{attribute 'call_after_init'}
FUNCTION_BLOCK FB_AmphosShutterEnable_Test EXTENDS FB_TestSuite
VAR_INPUT
END_VAR
VAR_OUTPUT
END_VAR
VAR
END_VAR

LocksWithHardwareFailure();
LocksWithLOCOLeak();
LocksWithLOTAOLeak();
LocksWithLUTLeak();
LocksWithAmphosOnAndTemperatureEvent01();
LocksWithAmphosOnAndTemperatureEvent02();
LocksWithAmphosOnAndTemperatureEvent03();
LocksWithAmphosOnAndTemperatureEvent04();
LocksWithTempMonError01();
LocksWithTempMonError02();
LocksWithTempMonError03();
LocksWithTempMonError04();
LocksWithTempMonError05();
LocksWithTempMonError06();
LocksWithTempMonError07();
LocksWithTempMonError08();
LocksWithOpcpaCriticalError();
LocksWithDumpChillerError();
LocksWithMRCError02();
LocksWithMRCError03();
EnablesWithAmphosOffAndTemperatureEvent01();
EnablesWithAmphosOffAndTemperatureEvent02();
EnablesWithAmphosOffAndTemperatureEvent03();
EnablesWithAmphosOffAndTemperatureEvent04();
EnablesWithTemperatureEventOverride01();
EnablesWithTemperatureEventOverride02();
EnablesWithTemperatureEventOverride03();
EnablesWithTemperatureEventOverride04();
EnablesWithOpcpaMinorError();
EnablesWhenNoError();

METHOD EnablesWhenNoError
VAR
	stErrors : st_ErrorStates;
	stOpcpaSetpoints : ST_LaserSetpoints := F_LaserSetpoints();
	bResult : BOOL;
END_VAR
TEST('EnablesWhenNoError');

bResult := F_AmphosShutterEnable(
	bAmphosOn := TRUE, 
	fOpcpaVoltage := stOpcpaSetpoints.nMinNominalVoltage, 
	bLoopTempOverride01 := FALSE,
	bLoopTempOverride02 := FALSE,
	bLoopTempOverride03 := FALSE,
	bLoopTempOverride04 := FALSE,
	stErrors := stErrors,
	stOpcpaSetpoints := stOpcpaSetpoints
);

AssertTrue(bResult, 'Amphos Shutter did not enable');

TEST_FINISHED();
END_METHOD

METHOD EnablesWithAmphosOffAndTemperatureEvent01
VAR
	stErrors : st_ErrorStates;
	stOpcpaSetpoints : ST_LaserSetpoints := F_LaserSetpoints();
	bResult : BOOL;
END_VAR
TEST('EnablesWithAmphosOffAndTemperatureEvent01');

stErrors.bChillerLoop01 := TRUE;
bResult := F_AmphosShutterEnable(
	bAmphosOn := FALSE, 
	fOpcpaVoltage := stOpcpaSetpoints.nMinNominalVoltage, 
	bLoopTempOverride01 := FALSE,
	bLoopTempOverride02 := FALSE,
	bLoopTempOverride03 := FALSE,
	bLoopTempOverride04 := FALSE,
	stErrors := stErrors,
	stOpcpaSetpoints := stOpcpaSetpoints
);

AssertTrue(bResult, 'Amphos Shutter did not enable');

TEST_FINISHED();
END_METHOD

METHOD EnablesWithAmphosOffAndTemperatureEvent02
VAR
	stErrors : st_ErrorStates;
	stOpcpaSetpoints : ST_LaserSetpoints := F_LaserSetpoints();
	bResult : BOOL;
END_VAR
TEST('EnablesWithAmphosOffAndTemperatureEvent02');

stErrors.bChillerLoop02 := TRUE;
bResult := F_AmphosShutterEnable(
	bAmphosOn := FALSE, 
	fOpcpaVoltage := stOpcpaSetpoints.nMinNominalVoltage, 
	bLoopTempOverride01 := FALSE,
	bLoopTempOverride02 := FALSE,
	bLoopTempOverride03 := FALSE,
	bLoopTempOverride04 := FALSE,
	stErrors := stErrors,
	stOpcpaSetpoints := stOpcpaSetpoints
);

AssertTrue(bResult, 'Amphos Shutter did not enable');

TEST_FINISHED();
END_METHOD

METHOD EnablesWithAmphosOffAndTemperatureEvent03
VAR
	stErrors : st_ErrorStates;
	stOpcpaSetpoints : ST_LaserSetpoints := F_LaserSetpoints();
	bResult : BOOL;
END_VAR
TEST('EnablesWithAmphosOffAndTemperatureEvent03');

stErrors.bChillerLoop03 := TRUE;
bResult := F_AmphosShutterEnable(
	bAmphosOn := FALSE, 
	fOpcpaVoltage := stOpcpaSetpoints.nMinNominalVoltage, 
	bLoopTempOverride01 := FALSE,
	bLoopTempOverride02 := FALSE,
	bLoopTempOverride03 := FALSE,
	bLoopTempOverride04 := FALSE,
	stErrors := stErrors,
	stOpcpaSetpoints := stOpcpaSetpoints
);

AssertTrue(bResult, 'Amphos Shutter did not enable');

TEST_FINISHED();
END_METHOD

METHOD EnablesWithAmphosOffAndTemperatureEvent04
VAR
	stErrors : st_ErrorStates;
	stOpcpaSetpoints : ST_LaserSetpoints := F_LaserSetpoints();
	bResult : BOOL;
END_VAR
TEST('EnablesWithAmphosOffAndTemperatureEvent04');

stErrors.bChillerLoop04 := TRUE;
bResult := F_AmphosShutterEnable(
	bAmphosOn := FALSE, 
	fOpcpaVoltage := stOpcpaSetpoints.nMinNominalVoltage, 
	bLoopTempOverride01 := FALSE,
	bLoopTempOverride02 := FALSE,
	bLoopTempOverride03 := FALSE,
	bLoopTempOverride04 := FALSE,
	stErrors := stErrors,
	stOpcpaSetpoints := stOpcpaSetpoints
);

AssertTrue(bResult, 'Amphos Shutter did not enable');

TEST_FINISHED();
END_METHOD

METHOD EnablesWithOpcpaMinorError
VAR
	stErrors : st_ErrorStates;
	stOpcpaSetpoints : ST_LaserSetpoints := F_LaserSetpoints();
	bResult : BOOL;
END_VAR
TEST('EnablesWithOpcpaMinorError');

stErrors.bOpcpaBeam := TRUE;
bResult := F_AmphosShutterEnable(
	bAmphosOn := TRUE, 
	fOpcpaVoltage := stOpcpaSetpoints.nMinNominalVoltage - 0.001, 
	bLoopTempOverride01 := FALSE,
	bLoopTempOverride02 := FALSE,
	bLoopTempOverride03 := FALSE,
	bLoopTempOverride04 := FALSE,
	stErrors := stErrors,
	stOpcpaSetpoints := stOpcpaSetpoints
);

AssertTrue(bResult, 'Amphos Shutter did not enable');

TEST_FINISHED();
END_METHOD

METHOD EnablesWithTemperatureEventOverride01
VAR
	stErrors : st_ErrorStates;
	stOpcpaSetpoints : ST_LaserSetpoints := F_LaserSetpoints();
	bResult : BOOL;
END_VAR
TEST('EnablesWithTemperatureEventOverride01');

stErrors.bChillerLoop01 := TRUE;
bResult := F_AmphosShutterEnable(
	bAmphosOn := TRUE, 
	fOpcpaVoltage := stOpcpaSetpoints.nMinNominalVoltage, 
	bLoopTempOverride01 := TRUE,
	bLoopTempOverride02 := FALSE,
	bLoopTempOverride03 := FALSE,
	bLoopTempOverride04 := FALSE,
	stErrors := stErrors,
	stOpcpaSetpoints := stOpcpaSetpoints
);

AssertTrue(bResult, 'Amphos Shutter did not enable');

TEST_FINISHED();
END_METHOD

METHOD EnablesWithTemperatureEventOverride02
VAR
	stErrors : st_ErrorStates;
	stOpcpaSetpoints : ST_LaserSetpoints := F_LaserSetpoints();
	bResult : BOOL;
END_VAR
TEST('EnablesWithTemperatureEventOverride02');

stErrors.bChillerLoop02 := TRUE;
bResult := F_AmphosShutterEnable(
	bAmphosOn := TRUE, 
	fOpcpaVoltage := stOpcpaSetpoints.nMinNominalVoltage, 
	bLoopTempOverride01 := FALSE,
	bLoopTempOverride02 := TRUE,
	bLoopTempOverride03 := FALSE,
	bLoopTempOverride04 := FALSE,
	stErrors := stErrors,
	stOpcpaSetpoints := stOpcpaSetpoints
);

AssertTrue(bResult, 'Amphos Shutter did not enable');

TEST_FINISHED();
END_METHOD

METHOD EnablesWithTemperatureEventOverride03
VAR
	stErrors : st_ErrorStates;
	stOpcpaSetpoints : ST_LaserSetpoints := F_LaserSetpoints();
	bResult : BOOL;
END_VAR
TEST('EnablesWithTemperatureEventOverride03');

stErrors.bChillerLoop03 := TRUE;
bResult := F_AmphosShutterEnable(
	bAmphosOn := TRUE, 
	fOpcpaVoltage := stOpcpaSetpoints.nMinNominalVoltage, 
	bLoopTempOverride01 := FALSE,
	bLoopTempOverride02 := FALSE,
	bLoopTempOverride03 := TRUE,
	bLoopTempOverride04 := FALSE,
	stErrors := stErrors,
	stOpcpaSetpoints := stOpcpaSetpoints
);

AssertTrue(bResult, 'Amphos Shutter did not enable');

TEST_FINISHED();
END_METHOD

METHOD EnablesWithTemperatureEventOverride04
VAR
	stErrors : st_ErrorStates;
	stOpcpaSetpoints : ST_LaserSetpoints := F_LaserSetpoints();
	bResult : BOOL;
END_VAR
TEST('EnablesWithTemperatureEventOverride04');

stErrors.bChillerLoop04 := TRUE;
bResult := F_AmphosShutterEnable(
	bAmphosOn := TRUE, 
	fOpcpaVoltage := stOpcpaSetpoints.nMinNominalVoltage, 
	bLoopTempOverride01 := FALSE,
	bLoopTempOverride02 := FALSE,
	bLoopTempOverride03 := FALSE,
	bLoopTempOverride04 := TRUE,
	stErrors := stErrors,
	stOpcpaSetpoints := stOpcpaSetpoints
);

AssertTrue(bResult, 'Amphos Shutter did not enable');

TEST_FINISHED();
END_METHOD

METHOD LocksWithAmphosOnAndTemperatureEvent01
VAR
	stErrors : st_ErrorStates;
	stOpcpaSetpoints : ST_LaserSetpoints := F_LaserSetpoints();
	bResult : BOOL;
END_VAR
TEST('LocksWithAmphosOnAndTemperatureEvent01');

stErrors.bChillerLoop01 := TRUE;
bResult := F_AmphosShutterEnable(
	bAmphosOn := TRUE, 
	fOpcpaVoltage := stOpcpaSetpoints.nMinNominalVoltage, 
	bLoopTempOverride01 := FALSE,
	bLoopTempOverride02 := FALSE,
	bLoopTempOverride03 := FALSE,
	bLoopTempOverride04 := FALSE,
	stErrors := stErrors,
	stOpcpaSetpoints := stOpcpaSetpoints
);

AssertFalse(bResult, 'Amphos Shutter did not lock');

TEST_FINISHED();
END_METHOD

METHOD LocksWithAmphosOnAndTemperatureEvent02
VAR
	stErrors : st_ErrorStates;
	stOpcpaSetpoints : ST_LaserSetpoints := F_LaserSetpoints();
	bResult : BOOL;
END_VAR
TEST('LocksWithAmphosOnAndTemperatureEvent02');

stErrors.bChillerLoop02 := TRUE;
bResult := F_AmphosShutterEnable(
	bAmphosOn := TRUE, 
	fOpcpaVoltage := stOpcpaSetpoints.nMinNominalVoltage, 
	bLoopTempOverride01 := FALSE,
	bLoopTempOverride02 := FALSE,
	bLoopTempOverride03 := FALSE,
	bLoopTempOverride04 := FALSE,
	stErrors := stErrors,
	stOpcpaSetpoints := stOpcpaSetpoints
);

AssertFalse(bResult, 'Amphos Shutter did not lock');

TEST_FINISHED();
END_METHOD

METHOD LocksWithAmphosOnAndTemperatureEvent03
VAR
	stErrors : st_ErrorStates;
	stOpcpaSetpoints : ST_LaserSetpoints := F_LaserSetpoints();
	bResult : BOOL;
END_VAR
TEST('LocksWithAmphosOnAndTemperatureEvent03');

stErrors.bChillerLoop03 := TRUE;
bResult := F_AmphosShutterEnable(
	bAmphosOn := TRUE, 
	fOpcpaVoltage := stOpcpaSetpoints.nMinNominalVoltage, 
	bLoopTempOverride01 := FALSE,
	bLoopTempOverride02 := FALSE,
	bLoopTempOverride03 := FALSE,
	bLoopTempOverride04 := FALSE,
	stErrors := stErrors,
	stOpcpaSetpoints := stOpcpaSetpoints
);

AssertFalse(bResult, 'Amphos Shutter did not lock');

TEST_FINISHED();
END_METHOD

METHOD LocksWithAmphosOnAndTemperatureEvent04
VAR
	stErrors : st_ErrorStates;
	stOpcpaSetpoints : ST_LaserSetpoints := F_LaserSetpoints();
	bResult : BOOL;
END_VAR
TEST('LocksWithAmphosOnAndTemperatureEvent04');

stErrors.bChillerLoop04 := TRUE;
bResult := F_AmphosShutterEnable(
	bAmphosOn := TRUE, 
	fOpcpaVoltage := stOpcpaSetpoints.nMinNominalVoltage, 
	bLoopTempOverride01 := FALSE,
	bLoopTempOverride02 := FALSE,
	bLoopTempOverride03 := FALSE,
	bLoopTempOverride04 := FALSE,
	stErrors := stErrors,
	stOpcpaSetpoints := stOpcpaSetpoints
);

AssertFalse(bResult, 'Amphos Shutter did not lock');

TEST_FINISHED();
END_METHOD

METHOD LocksWithDumpChillerError
VAR
	stErrors : st_ErrorStates;
	stOpcpaSetpoints : ST_LaserSetpoints := F_LaserSetpoints();
	bResult : BOOL;
END_VAR
TEST('LocksWithDumpChillerError');

stErrors.bDumpChiller := TRUE;
bResult := F_AmphosShutterEnable(
	bAmphosOn := TRUE, 
	fOpcpaVoltage := stOpcpaSetpoints.nMinNominalVoltage, 
	bLoopTempOverride01 := FALSE,
	bLoopTempOverride02 := FALSE,
	bLoopTempOverride03 := FALSE,
	bLoopTempOverride04 := FALSE,
	stErrors := stErrors,
	stOpcpaSetpoints := stOpcpaSetpoints
);

AssertFalse(bResult, 'Amphos Shutter did not lock');

TEST_FINISHED();
END_METHOD

METHOD LocksWithHardwareFailure
VAR
	stErrors : st_ErrorStates;
	stOpcpaSetpoints : ST_LaserSetpoints := F_LaserSetpoints();
	bResult : BOOL;
END_VAR
TEST('LocksWithHardwareFailure');

stErrors.bHardwareFailure := TRUE;
bResult := F_AmphosShutterEnable(
	bAmphosOn := TRUE, 
	fOpcpaVoltage := stOpcpaSetpoints.nMinNominalVoltage, 
	bLoopTempOverride01 := FALSE,
	bLoopTempOverride02 := FALSE,
	bLoopTempOverride03 := FALSE,
	bLoopTempOverride04 := FALSE,
	stErrors := stErrors,
	stOpcpaSetpoints := stOpcpaSetpoints
);

AssertFalse(bResult, 'Amphos Shutter did not lock');

TEST_FINISHED();
END_METHOD

METHOD LocksWithLOCOLeak
VAR
	stErrors : st_ErrorStates;
	stOpcpaSetpoints : ST_LaserSetpoints := F_LaserSetpoints();
	bResult : BOOL;
END_VAR
TEST('LocksWithLOCOLeak');

stErrors.bLeakOpcpaCarbideOn := TRUE;
bResult := F_AmphosShutterEnable(
	bAmphosOn := TRUE, 
	fOpcpaVoltage := stOpcpaSetpoints.nMinNominalVoltage, 
	bLoopTempOverride01 := FALSE,
	bLoopTempOverride02 := FALSE,
	bLoopTempOverride03 := FALSE,
	bLoopTempOverride04 := FALSE,
	stErrors := stErrors,
	stOpcpaSetpoints := stOpcpaSetpoints
);

AssertFalse(bResult, 'Amphos Shutter did not lock');

TEST_FINISHED();
END_METHOD

METHOD LocksWithLOTAOLeak
VAR
	stErrors : st_ErrorStates;
	stOpcpaSetpoints : ST_LaserSetpoints := F_LaserSetpoints();
	bResult : BOOL;
END_VAR
TEST('LocksWithLOTAOLeak');

stErrors.bLeakOpticalTableAmphosOn := TRUE;
bResult := F_AmphosShutterEnable(
	bAmphosOn := TRUE, 
	fOpcpaVoltage := stOpcpaSetpoints.nMinNominalVoltage, 
	bLoopTempOverride01 := FALSE,
	bLoopTempOverride02 := FALSE,
	bLoopTempOverride03 := FALSE,
	bLoopTempOverride04 := FALSE,
	stErrors := stErrors,
	stOpcpaSetpoints := stOpcpaSetpoints
);

AssertFalse(bResult, 'Amphos Shutter did not lock');

TEST_FINISHED();
END_METHOD

METHOD LocksWithLUTLeak
VAR
	stErrors : st_ErrorStates;
	stOpcpaSetpoints : ST_LaserSetpoints := F_LaserSetpoints();
	bResult : BOOL;
END_VAR
TEST('LocksWithLUTLeak');

stErrors.bLeakUnderTable := TRUE;
bResult := F_AmphosShutterEnable(
	bAmphosOn := TRUE, 
	fOpcpaVoltage := stOpcpaSetpoints.nMinNominalVoltage, 
	bLoopTempOverride01 := FALSE,
	bLoopTempOverride02 := FALSE,
	bLoopTempOverride03 := FALSE,
	bLoopTempOverride04 := FALSE,
	stErrors := stErrors,
	stOpcpaSetpoints := stOpcpaSetpoints
);

AssertFalse(bResult, 'Amphos Shutter did not lock');

TEST_FINISHED();
END_METHOD

METHOD LocksWithMRCError02
VAR
	stErrors : st_ErrorStates;
	stOpcpaSetpoints : ST_LaserSetpoints := F_LaserSetpoints();
	bResult : BOOL;
END_VAR
TEST('LocksWithMRCError02');

stErrors.bAmphosMRC02 := TRUE;
bResult := F_AmphosShutterEnable(
	bAmphosOn := TRUE, 
	fOpcpaVoltage := stOpcpaSetpoints.nMinNominalVoltage, 
	bLoopTempOverride01 := FALSE,
	bLoopTempOverride02 := FALSE,
	bLoopTempOverride03 := FALSE,
	bLoopTempOverride04 := FALSE,
	stErrors := stErrors,
	stOpcpaSetpoints := stOpcpaSetpoints
);

AssertFalse(bResult, 'Amphos Shutter did not lock');

TEST_FINISHED();
END_METHOD

METHOD LocksWithMRCError03
VAR
	stErrors : st_ErrorStates;
	stOpcpaSetpoints : ST_LaserSetpoints := F_LaserSetpoints();
	bResult : BOOL;
END_VAR
TEST('LocksWithMRCError03');

stErrors.bAmphosMRC03 := TRUE;
bResult := F_AmphosShutterEnable(
	bAmphosOn := TRUE, 
	fOpcpaVoltage := stOpcpaSetpoints.nMinNominalVoltage, 
	bLoopTempOverride01 := FALSE,
	bLoopTempOverride02 := FALSE,
	bLoopTempOverride03 := FALSE,
	bLoopTempOverride04 := FALSE,
	stErrors := stErrors,
	stOpcpaSetpoints := stOpcpaSetpoints
);

AssertFalse(bResult, 'Amphos Shutter did not lock');

TEST_FINISHED();
END_METHOD

METHOD LocksWithOpcpaCriticalError
VAR
	stErrors : st_ErrorStates;
	stOpcpaSetpoints : ST_LaserSetpoints := F_LaserSetpoints();
	bResult : BOOL;
END_VAR
TEST('LocksWithOpcpaCriticalError');

stErrors.bOpcpaBeam := TRUE;
bResult := F_AmphosShutterEnable(
	bAmphosOn := TRUE, 
	fOpcpaVoltage := stOpcpaSetpoints.nMinVoltage - 1, 
	bLoopTempOverride01 := FALSE,
	bLoopTempOverride02 := FALSE,
	bLoopTempOverride03 := FALSE,
	bLoopTempOverride04 := FALSE,
	stErrors := stErrors,
	stOpcpaSetpoints := stOpcpaSetpoints
);

AssertFalse(bResult, 'Amphos Shutter did not lock');

TEST_FINISHED();
END_METHOD

METHOD LocksWithTempMonError01
VAR
	stErrors : st_ErrorStates;
	stOpcpaSetpoints : ST_LaserSetpoints := F_LaserSetpoints();
	bResult : BOOL;
END_VAR
TEST('LocksWithTempMonError01');

stErrors.bTempMon01 := TRUE;
bResult := F_AmphosShutterEnable(
	bAmphosOn := TRUE, 
	fOpcpaVoltage := stOpcpaSetpoints.nMinNominalVoltage, 
	bLoopTempOverride01 := FALSE,
	bLoopTempOverride02 := FALSE,
	bLoopTempOverride03 := FALSE,
	bLoopTempOverride04 := FALSE,
	stErrors := stErrors,
	stOpcpaSetpoints := stOpcpaSetpoints
);

AssertFalse(bResult, 'Amphos Shutter did not lock');

TEST_FINISHED();
END_METHOD

METHOD LocksWithTempMonError02
VAR
	stErrors : st_ErrorStates;
	stOpcpaSetpoints : ST_LaserSetpoints := F_LaserSetpoints();
	bResult : BOOL;
END_VAR
TEST('LocksWithTempMonError02');

stErrors.bTempMon02 := TRUE;
bResult := F_AmphosShutterEnable(
	bAmphosOn := TRUE, 
	fOpcpaVoltage := stOpcpaSetpoints.nMinNominalVoltage, 
	bLoopTempOverride01 := FALSE,
	bLoopTempOverride02 := FALSE,
	bLoopTempOverride03 := FALSE,
	bLoopTempOverride04 := FALSE,
	stErrors := stErrors,
	stOpcpaSetpoints := stOpcpaSetpoints
);

AssertFalse(bResult, 'Amphos Shutter did not lock');

TEST_FINISHED();
END_METHOD

METHOD LocksWithTempMonError03
VAR
	stErrors : st_ErrorStates;
	stOpcpaSetpoints : ST_LaserSetpoints := F_LaserSetpoints();
	bResult : BOOL;
END_VAR
TEST('LocksWithTempMonError03');

stErrors.bTempMon03 := TRUE;
bResult := F_AmphosShutterEnable(
	bAmphosOn := TRUE, 
	fOpcpaVoltage := stOpcpaSetpoints.nMinNominalVoltage, 
	bLoopTempOverride01 := FALSE,
	bLoopTempOverride02 := FALSE,
	bLoopTempOverride03 := FALSE,
	bLoopTempOverride04 := FALSE,
	stErrors := stErrors,
	stOpcpaSetpoints := stOpcpaSetpoints
);

AssertFalse(bResult, 'Amphos Shutter did not lock');

TEST_FINISHED();
END_METHOD

METHOD LocksWithTempMonError04
VAR
	stErrors : st_ErrorStates;
	stOpcpaSetpoints : ST_LaserSetpoints := F_LaserSetpoints();
	bResult : BOOL;
END_VAR
TEST('LocksWithTempMonError04');

stErrors.bTempMon04 := TRUE;
bResult := F_AmphosShutterEnable(
	bAmphosOn := TRUE, 
	fOpcpaVoltage := stOpcpaSetpoints.nMinNominalVoltage, 
	bLoopTempOverride01 := FALSE,
	bLoopTempOverride02 := FALSE,
	bLoopTempOverride03 := FALSE,
	bLoopTempOverride04 := FALSE,
	stErrors := stErrors,
	stOpcpaSetpoints := stOpcpaSetpoints
);

AssertFalse(bResult, 'Amphos Shutter did not lock');

TEST_FINISHED();
END_METHOD

METHOD LocksWithTempMonError05
VAR
	stErrors : st_ErrorStates;
	stOpcpaSetpoints : ST_LaserSetpoints := F_LaserSetpoints();
	bResult : BOOL;
END_VAR
TEST('LocksWithTempMonError05');

stErrors.bTempMon05 := TRUE;
bResult := F_AmphosShutterEnable(
	bAmphosOn := TRUE, 
	fOpcpaVoltage := stOpcpaSetpoints.nMinNominalVoltage, 
	bLoopTempOverride01 := FALSE,
	bLoopTempOverride02 := FALSE,
	bLoopTempOverride03 := FALSE,
	bLoopTempOverride04 := FALSE,
	stErrors := stErrors,
	stOpcpaSetpoints := stOpcpaSetpoints
);

AssertFalse(bResult, 'Amphos Shutter did not lock');

TEST_FINISHED();
END_METHOD

METHOD LocksWithTempMonError06
VAR
	stErrors : st_ErrorStates;
	stOpcpaSetpoints : ST_LaserSetpoints := F_LaserSetpoints();
	bResult : BOOL;
END_VAR
TEST('LocksWithTempMonError06');

stErrors.bTempMon06 := TRUE;
bResult := F_AmphosShutterEnable(
	bAmphosOn := TRUE, 
	fOpcpaVoltage := stOpcpaSetpoints.nMinNominalVoltage, 
	bLoopTempOverride01 := FALSE,
	bLoopTempOverride02 := FALSE,
	bLoopTempOverride03 := FALSE,
	bLoopTempOverride04 := FALSE,
	stErrors := stErrors,
	stOpcpaSetpoints := stOpcpaSetpoints
);

AssertFalse(bResult, 'Amphos Shutter did not lock');

TEST_FINISHED();
END_METHOD

METHOD LocksWithTempMonError07
VAR
	stErrors : st_ErrorStates;
	stOpcpaSetpoints : ST_LaserSetpoints := F_LaserSetpoints();
	bResult : BOOL;
END_VAR
TEST('LocksWithTempMonError07');

stErrors.bTempMon07 := TRUE;
bResult := F_AmphosShutterEnable(
	bAmphosOn := TRUE, 
	fOpcpaVoltage := stOpcpaSetpoints.nMinNominalVoltage, 
	bLoopTempOverride01 := FALSE,
	bLoopTempOverride02 := FALSE,
	bLoopTempOverride03 := FALSE,
	bLoopTempOverride04 := FALSE,
	stErrors := stErrors,
	stOpcpaSetpoints := stOpcpaSetpoints
);

AssertFalse(bResult, 'Amphos Shutter did not lock');

TEST_FINISHED();
END_METHOD

METHOD LocksWithTempMonError08
VAR
	stErrors : st_ErrorStates;
	stOpcpaSetpoints : ST_LaserSetpoints := F_LaserSetpoints();
	bResult : BOOL;
END_VAR
TEST('LocksWithTempMonError08');

stErrors.bTempMon08 := TRUE;
bResult := F_AmphosShutterEnable(
	bAmphosOn := TRUE, 
	fOpcpaVoltage := stOpcpaSetpoints.nMinNominalVoltage, 
	bLoopTempOverride01 := FALSE,
	bLoopTempOverride02 := FALSE,
	bLoopTempOverride03 := FALSE,
	bLoopTempOverride04 := FALSE,
	stErrors := stErrors,
	stOpcpaSetpoints := stOpcpaSetpoints
);

AssertFalse(bResult, 'Amphos Shutter did not lock');

TEST_FINISHED();
END_METHOD

END_FUNCTION_BLOCK

(* stored: Version 1.1.0.1, ProductVersion 3.1.4022.17
   POU FB_AmphosShutterEnable_Test: Id {003c19f0-18c9-4e63-8c2d-0d1529cf21e6}, SpecialFunc None
   Method EnablesWhenNoError: Id {073e45da-bab5-4ad7-ba6c-e7e3d3582e6b}
   Method EnablesWithAmphosOffAndTemperatureEvent01: Id {6b254004-17be-4ccd-bff4-6ed05457aecc}
   Method EnablesWithAmphosOffAndTemperatureEvent02: Id {0b69e9f4-9eca-4fe3-a56b-09838e2d815d}
   Method EnablesWithAmphosOffAndTemperatureEvent03: Id {ac4627a4-aab9-4c34-8899-1f167dc7e06a}
   Method EnablesWithAmphosOffAndTemperatureEvent04: Id {23ec8852-e2d8-4329-866c-f1226e7e901e}
   Method EnablesWithOpcpaMinorError: Id {fd881f51-9c28-4e11-8800-5f27f02870db}
   Method EnablesWithTemperatureEventOverride01: Id {ece501f0-c578-4b02-80e9-cb4721d8b6d5}
   Method EnablesWithTemperatureEventOverride02: Id {d4c7792e-1f61-417b-aeeb-1057d2498c55}
   Method EnablesWithTemperatureEventOverride03: Id {93a87445-6cf1-4dba-bde8-dd5cf9a68c17}
   Method EnablesWithTemperatureEventOverride04: Id {d1f00ddc-a889-4939-915e-2768ec4cf363}
   Method LocksWithAmphosOnAndTemperatureEvent01: Id {662b51f8-8f66-4fbf-bb56-1241734e69d9}
   Method LocksWithAmphosOnAndTemperatureEvent02: Id {236cabca-1ab4-4b17-97a8-e591567c64fb}
   Method LocksWithAmphosOnAndTemperatureEvent03: Id {5745d4f0-3bf8-4b37-92b3-87d0a40e2b85}
   Method LocksWithAmphosOnAndTemperatureEvent04: Id {e872d4ae-7049-4674-9e30-25b2069f30e8}
   Method LocksWithDumpChillerError: Id {6aef82c6-6293-4c61-b609-5c9371e3e53b}
   Method LocksWithHardwareFailure: Id {a42f0405-354a-4b42-90c7-b52d9dc9cf21}
   Method LocksWithLOCOLeak: Id {91dd1cee-ab35-4242-af87-11f34e00c99b}
   Method LocksWithLOTAOLeak: Id {72405b24-2bcc-4d93-a3ae-f702e92929cd}
   Method LocksWithLUTLeak: Id {a04eef41-8280-4c52-9b8d-74bedfe2bdbc}
   Method LocksWithMRCError02: Id {26e46157-21ae-4473-828b-31afc1338e16}
   Method LocksWithMRCError03: Id {4bdcf774-43ac-4b27-8480-469e007c397f}
   Method LocksWithOpcpaCriticalError: Id {c17b86f8-025b-4320-a4b5-7331a7f9f5a9}
   Method LocksWithTempMonError01: Id {90bd4956-9c90-4069-93be-d3d9bf695bf9}
   Method LocksWithTempMonError02: Id {69ff6c56-5168-4f7d-b6b7-b6b4d864cfed}
   Method LocksWithTempMonError03: Id {33187f00-3335-491e-827f-e095cf24a5a7}
   Method LocksWithTempMonError04: Id {9280837d-f10b-4a13-959f-9459ccd5076b}
   Method LocksWithTempMonError05: Id {a3b8cb22-10a1-49c7-af15-27a746f22d9a}
   Method LocksWithTempMonError06: Id {bcdd067a-2439-4556-8284-f79fa30c19ed}
   Method LocksWithTempMonError07: Id {b3cc9b9b-59ef-4db0-854d-66f239421b0c}
   Method LocksWithTempMonError08: Id {fb72dc15-3b01-46db-8fd8-cdd9a8c4166e} *)
